(* Logix 5000 project; controller Timers Emulate 5570 rev 33.11; software revision 33.00 *)

TASK T00_MainTask (continuous, watchdog 500 ms) : P00_MainProgram

MODULES
   Local : Emulate 5570 (ICP 2, rev 33.11)
END_MODULES

PROGRAM P00_MainProgram   (* main routine R00_MainRoutine *)
VAR
   ES : BOOL;   // Boton de Paro de emergencia
   O01_Lampara : BOOL;   // Luz de seguridad
   S01_Movimiento : BOOL;   // Sensor de Movimiento
   T01_DesactivarLuz : TIMER := (PRE := 10000);   // Timer para desactivar luz en 10s
END_VAR

ROUTINE R00_MainRoutine   (* ladder *)
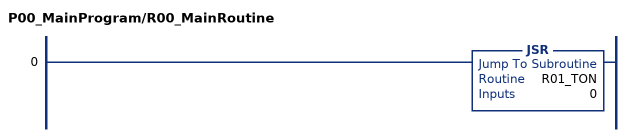
   0: JSR(R01_TON,0);
END_ROUTINE

ROUTINE R01_TON   (* ladder *)
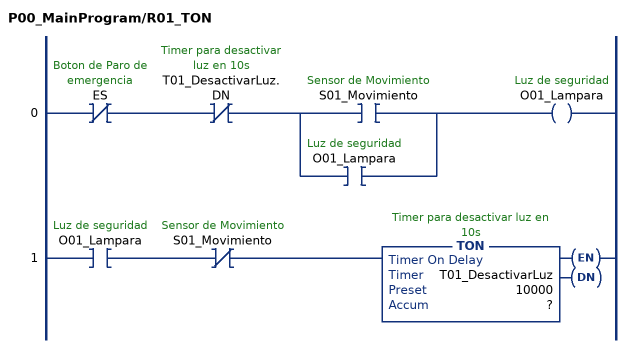
   0: XIO(ES)XIO(T01_DesactivarLuz.DN)[XIC(S01_Movimiento) ,XIC(O01_Lampara) ]OTE(O01_Lampara);
   1: XIC(O01_Lampara)XIO(S01_Movimiento)TON(T01_DesactivarLuz,?,?);
END_ROUTINE
END_PROGRAM
